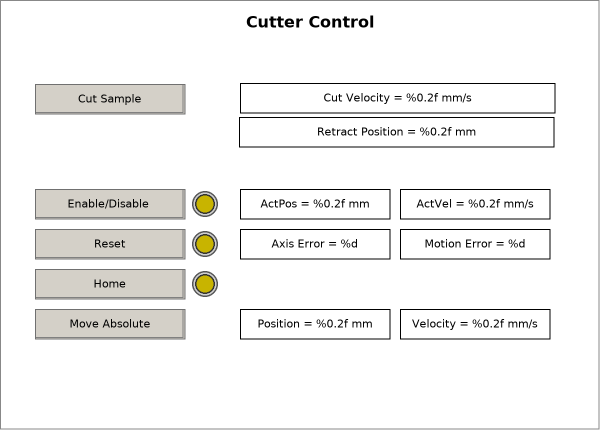
VISUALIZATION Manual_Cutter  // 600x430
    Label (133,7 355x30), "Cutter Control"
    Button (35,84 150x30), "Cut Sample", input disabled if: MAIN.fbSlitter.bBusy
        OnMouseClick: execute { MAIN.fbSlitter.Manual.bCutSample := TRUE; }
    Button (35,189 150x30), "Enable/Disable", input disabled if: MAIN.fbSlitter.bBusy
        OnMouseClick: execute { MAIN.fbSlitter.Manual.bCutterDisable := TRUE; }
    Button (35,229 150x30), "Reset", input disabled if: MAIN.fbSlitter.bBusy
        OnMouseClick: execute { MAIN.fbSlitter.Manual.bCutterReset := TRUE; }
    Button (35,269 150x30), "Home"
        OnMouseClick: execute { MAIN.fbSlitter.Manual.bCutterHome := TRUE; }
    Lamp1 (190,189 30x30), variable: MAIN.fbSlitter.Cutter.Axis.NcToPlc.StateDWord.0 = 1, style: Lamp-Lamp1-Yellow
    Rectangle (240,229 150x30), "Axis Error = %d", text variable: MAIN.fbSlitter.Cutter.Axis.NcToPlc.ErrorCode
    Lamp1 (190,229 30x30), variable: MAIN.fbSlitter.Cutter.Axis.NcToPlc.ErrorCode <> 0, style: Lamp-Lamp1-Yellow
    Lamp1 (190,269 30x30), variable: MAIN.fbSlitter.Cutter.Axis.NcToPlc.StateDWord.1 = 1, style: Lamp-Lamp1-Yellow
    Rectangle (400,229 150x30), "Motion Error = %d", text variable: MAIN.fbSlitter.Cutter._errorCode
    Button (35,309 150x30), "Move Absolute"
        OnMouseClick: execute { MAIN.fbSlitter.Manual.bCutterMoveAbs := TRUE; }
    Rectangle (240,309 150x30), "Position = %0.2f mm", text variable: MAIN.fbSlitter.Cutter._position
        OnMouseClick: write MAIN.fbSlitter.Cutter._position via Default, min 0, max 20, title 'Cutter Position'
    Rectangle (400,309 150x30), "Velocity = %0.2f mm/s", text variable: MAIN.fbSlitter.Cutter._velocity
        OnMouseClick: write MAIN.fbSlitter.Cutter._velocity via Default, title 'Cutter Velocity'
    Rectangle (240,189 150x30), "ActPos = %0.2f mm", text variable: MAIN.fbSlitter.Cutter.Axis.NcToPlc.ActPos
    Rectangle (400,189 150x30), "ActVel = %0.2f mm/s", text variable: MAIN.fbSlitter.Cutter.Axis.NcToPlc.ActVelo
    Rectangle (240,83 315x30), "Cut Velocity = %0.2f mm/s", text variable: MAIN.fbSlitter.Cutter._hmiParameters.cutVelocity
        OnMouseClick: write MAIN.fbSlitter.Cutter._hmiParameters.cutVelocity via Default, title 'Cutter Velocity'
    Rectangle (239,117 315x30), "Retract Position = %0.2f mm", text variable: MAIN.fbSlitter.Cutter._hmiParameters.retractPosition
        OnMouseClick: write MAIN.fbSlitter.Cutter._hmiParameters.retractPosition via Default, title 'Retract Position'
END_VISUALIZATION

(* stored: Version 1.1.0.1, ProductVersion 3.1.4024.9
   Visu Manual_Cutter: Id {7587e01b-fbe4-408d-9c69-57394852caaa} *)
